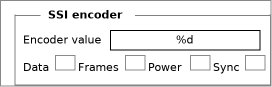
VISUALIZATION VISU_SSIEncoder  // 272x87
VAR_IN_OUT
	ref : SSIEncoder;
END_VAR
    Polyline (135,15) (270,15) (270,85) (15,85) (15,15) (40,15)
    Label (45,5 150x20), "SSI encoder"
    Rectangle (110,30 150x20), "%d", text variable: ref.counterValue
    Label (20,55 40x25), "Data"
    Frame (55,55 20x15)
        shows VISU_State_green_red(state := ref.dataError)
    Frame (125,55 20x15)
        shows VISU_State_green_red(state := ref.frameError)
    Label (75,55 50x25), "Frames"
    Label (145,55 45x25), "Power"
    Frame (190,55 20x15)
        shows VISU_State_green_red(state := ref.powerFailure)
    Frame (245,55 20x15)
        shows VISU_State_green_red(state := ref.syncError)
    Label (210,55 35x25), "Sync"
    Label (20,30 90x20), "Encoder value"
END_VISUALIZATION

(* stored: Version 1.1.0.1, ProductVersion 3.1.4019.2
   Visu VISU_SSIEncoder: Id {bba2b667-3254-4e00-8825-1b27fb1195c8} *)
